TYPE EM_Transport_PAR :
STRUCT
END_STRUCT
END_TYPE

(* stored: Version 1.1.0.1, ProductVersion 3.1.4024.12
   DUT EM_Transport_PAR: Id {be6e383e-f27e-4208-bbaf-2431509631d5} *)
